(* CoDeSys 2.3 export: MONTH_TO_STRING.EXP *)

(* POU String/MONTH_TO_STRING, ST *)
FUNCTION MONTH_TO_STRING : STRING(10)
VAR_INPUT
	MTH : INT;
	LANG : INT;
	LX : INT;
END_VAR
VAR
	ly : INT;
END_VAR

(*
version 1.1	19. oct. 2008
programmer 	hugo
tested by	oscat

MONTH_TO_STRING converts an Integer 1..12 into a String with the Names of the corresponding Month.
the decoding is according to the language setup in global vars

*)
IF LANG = 0 THEN Ly := LANGUAGE.DEFAULT; ELSE ly := MIN(LANG, language.LMAX); END_IF;
IF MTH < 1 OR MTH > 12 THEN
	RETURN;
ELSIF LX = 0 THEN
	MONTH_TO_STRING := language.MONTHS[ly, MTH];
ELSIF Lx = 3 THEN
	MONTH_TO_STRING := language.MONTHS3[ly, MTH];
END_IF;


(* revisison history

hm	21. sep. 2008	rev 1.0
	original version

hm	19. oct. 2008	rev 1.1
	changed language setup constants
*)
END_FUNCTION
